PROGRAM PRG_SIMULATION
VAR
END_VAR

// valves

fbVgc_TV2K4_VGC_1(
	stAVol := stVl_Start,
	stBvol := stVl_Proto,
	stValve := stVgc_TV2K4_VGC_1
	); // VV9S
	
fbVgc_MR1K4_VGC_1(
	stAVol := stVl_Proto,
	stBvol := stVl_End,
	stValve := stVgc_MR1K4_VGC_1
	); // VV10S

// gauges

fbMks275_TV2K4_GPI_1(stVolume := stVl_Proto, stGauge:= stMks275_TV2K4_GPI_1);
fbMks500_TV2K4_GCC_1(stVolume := stVl_Proto, stGauge:= stMks500_TV2K4_GCC_1);

// pumps

fbGamPip_TV2KO_PIP_1(stVolume := stVl_Proto, stPip := stGamPip_TV2KO_PIP_1);

END_PROGRAM

(* stored: Version 1.1.0.1, ProductVersion 3.1.4022.12
   POU PRG_SIMULATION: Id {ec1bb7bb-e266-4a42-8f10-1901cc9e9ecf}, SpecialFunc None *)
